% RSLogix 500 project WFETC_TOTS_R0.RSS, saved by version 12.00.00.00 %
PROJECT "WFETC"    % processor: SLC 500, 1747-L552 %

PROGRAM FILES
  LAD 2 "MAIN"  23 rungs
  LAD 3 "TE CONTROL"  1 rungs  % Set NT4 Input modules for Type J T/C's and °C Unit %
  LAD 4 "RIO BTRWS"  15 rungs  % Block Transfers for Remote IO %
  LAD 10 "ALARM CTRL"  9 rungs  % Alarm Controls %
  LAD 11 "ALARMS"  53 rungs  % Process Alarms %
  LAD 15 "IFIX PBS"  8 rungs  % iFIX PBs %
  LAD 16 "PV PBS"  11 rungs  % Panel View Screen Movement PB's %
  LAD 17 "VFD USERS"  17 rungs  % Determines which user is using each VFD %
  LAD 31 "MOVE TES"  20 rungs  % Move TE Info to Sequencial Locations, etc %
  LAD 32 "MOVE PTS"  7 rungs  % Move PT Info to Sequencial Locations, etc %
  LAD 33 "MOVE FTS"  6 rungs  % Move FT Info to Sequencial Locations, etc %
  LAD 34 "CALC WTS"  9 rungs  % Convert Remote I/O Data to Real Data for All Scale %
  LAD 35 "CALC WT FT"  10 rungs  % Calcualte Flow Rates based on Weight Changes %
  LAD 36 "CALC PTS"  15 rungs  % Calculate PT's Based on Max & Min Ranges %
  LAD 37 "CALC FTS"  8 rungs  % Calculate FT's Based on Max & Min Ranges %
  LAD 38 "CALC FYS"  35 rungs  % Calculate Flow Rates based on Scale Change & Time %
  LAD 39 "CALC ITS"  10 rungs  % Calculate SY Current Values %
  LAD 40 "CALC ATS"  7 rungs  % Calculate Densitys from FlowMeters %
  LAD 41 "CAL FTAVGS"  7 rungs  % Calculate FT Averages %
  LAD 42 "CALC LITS"  2 rungs  % Calculate LIT values %
  LAD 43 "CALLC TITS"  2 rungs  % Calculate TITs %
  LAD 48 "EF-1"  8 rungs  % Process Area Exhaust Fan Controls %
  LAD 49 "EF-2"  8 rungs  % Utility Room Exhaust Fan Controls %
  LAD 50 "EV-01"  8 rungs  % EV-1 Rotor Controls %
  LAD 51 "EV-02"  12 rungs  % EV-2 Rotor Drive VFD Controls %
  LAD 52 "EV-03"  12 rungs  % EV-3 Rotor Drive VFD Controls %
  LAD 53 "AG-04"  12 rungs  % AG-4 Agitator Drive VFD Controls %
  LAD 56 "VP-09"  8 rungs  % VP-9 Beach-Ross Vacuum Pump Controls %
  LAD 57 "VP-10"  8 rungs  % VP-10 Kinney Vacuum Pump Controls %
  LAD 60 "PU-11"  8 rungs  % PU-11 Tempered Water Loop No-1 Circ Pump Controls %
  LAD 61 "PU-12"  8 rungs  % PU-12 Tempered Water Loop No-2 Circ Pump Controls %
  LAD 62 "PU-15"  8 rungs  % PU-15 Tempered Oil Loop No-1 Circ Pump Controls %
  LAD 63 "EV-20"  12 rungs  % EV-20 Rotor Drive VFD Controls %
  LAD 64 "PU-21-1"  11 rungs  % PU-21-1 Feed Pump No-1 Controls %
  LAD 65 "PU-21-2"  11 rungs  % PU-21-2 Feed Pump No-2 Controls %
  LAD 66 "PU-21-3"  11 rungs  % PU-21-3 Feed Pump No-3 Controls %
  LAD 67 "PU-21-4"  11 rungs  % PU-21-4 Feed Pump No-4 Controls %
  LAD 69 "PU-22-1"  11 rungs  % PU-22-1 Level Pump No-1 Controls %
  LAD 71 "PU-23"  10 rungs  % PU-23 Hot Oil Circ Pump Controls %
  LAD 72 "EH-24"  7 rungs  % EH-24 Hot Oil Heater Controls %
  LAD 73 "VB-26"  9 rungs  % VB-26 Beach-Ross Vacuum Blower Controls %
  LAD 74 "PU-30"  9 rungs  % PU-30 Cooling Water Header Booster Pump Controls %
  LAD 75 "VB-35"  8 rungs  % VB-35 Tuthill Vacuum Blower Controls %
  LAD 77 "PU-37"  8 rungs  % PU-37, Temperaed Oil No-3 Controls %
  LAD 80 "PU-40"  8 rungs  % PU-40, Temperaed Oil No-2 Controls %
  LAD 81 "EV-42"  12 rungs  % EV-42 Rotor Drive VFD Controls %
  LAD 82 "PU-46"  11 rungs  % PU-46, Flash Evaporator Circ Pump %
  LAD 86 "ALL VFDS"  10 rungs  % Control All VFD's %
  LAD 90 "ALL PIDS"  17 rungs  % Execute All PID Statements using STI Interupt %
  LAD 101 "FIC-21-1"  12 rungs  % Feed Flow No-1 PID Controls %
  LAD 102 "FIC-21-2"  12 rungs  % Feed Flow No-2 PID Controls %
  LAD 103 "FIC-21-3"  12 rungs  % Feed Flow No-3 PID Controls %
  LAD 104 "FIC-21-4"  12 rungs  % Feed Flow No-4 PID Controls %
  LAD 111 "PIC-9-1"  14 rungs  % Vacuum Control No-1 PID %
  LAD 112 "PID-10-1"  14 rungs  % Vacuum Control No-2 PID %
  LAD 115 "PIC-28-1"  5 rungs  % Steam Pressure PID Controls %
  LAD 116 "PIC-30-1"  6 rungs  % Cooling Water Pressure PID Controls %
  LAD 117 "PIC-46-1"  6 rungs  % Flash Evap Pressure Controller %
  LAD 121 "TIC-11-1"  6 rungs  % Tempered Water Loop No-1 Temperature PID Controls %
  LAD 122 "TIC-12-1"  7 rungs  % Tempered Water Loop No-2 Temperature PID Controls %
  LAD 123 "TIC-15-1"  6 rungs  % Tempered Oil Loop No-1 Temperature PID Controls %
  LAD 124 "TIC-24-1"  6 rungs  % Hot Oil Temperature PID Controls %
  LAD 125 "TIC-37-1"  6 rungs  % Tempered Oil Loop No-3 Temperature PID Controls %
  LAD 126 "TIC-40-1"  6 rungs  % Tempered Oil Loop No-2 Temperature PID Controls %
  LAD 131 "LIC-22-1"  7 rungs  % Level Control No-1 PID Controls %
  LAD 132 "TOTALIZER"  8 rungs

DATA FILES
  O0 OUTPUT  99 elements
  I1 INPUT  111 elements
  S2 STATUS  83 elements
  B3 BINARY  81 elements
  T4 TIMER  36 elements
  C5 COUNTER  15 elements
  R6 CONTROL  1 elements
  N7 INTEGER  23 elements
  F8 FLOAT  256 elements
  N11 AI INTEGER  250 elements  % Integer Data for All Inputs (TE's, PT's and FT's) %
  N12 RIO DATA  200 elements  % Remote I/O Data %
  N13 TE SETUP  200 elements  % TE Setup Data %
  F14 SETPOINTS  100 elements  % Setpoints for various Alarms, trips, etc %
  N15 PID 1 OF 3  240 elements  % PID Statement Controls File No-1 %
  N16 PID 2 OF 3  175 elements  % PID Statement Controls File No-2 %
  N17 PID 3 OF 3  180 elements  % PID Statement Controls File No-3 %
  N18 PID OUTPUT  60 elements  % Outputs from All PID Statements %
  N20 PANELVIEW  100 elements  % Info From/to PanelView HMIs %
  F21 AI REAL  256 elements
  F22 AI BY TAG  250 elements
  N23 AI PTRS  256 elements
  N24 FIXED INTS  250 elements  % Fixed Integer Values %
  N25 VAR INTS  200 elements  % Variable Integer Values %
  F26 FIXEDREAL1  250 elements  % Fixed Real (Floating Point) Data 1 of 2 %
  F27 VAR REAL  210 elements  % Variable Real (Floatinf Point) Data %
  F28 FLOW AVGS  51 elements  % Flow Data used to Calculate 5 Minute Aveerages %
  F29 PID PCNTS1  250 elements  % PID Statement 0, 25, 50, 75 & 100% Values %
  F30 FIXEDREAL2  250 elements  % Fixed Real (Floating Point) Data 2 of 2 %
  F31 PID PCNTS2  220 elements
  N50 CNTL BITS  50 elements  % Control Bits for all Motors, Contacters, Etc %
  T51 ALARM TMRS  100 elements  % Alarm Timers %
  F52 ALARM SPS  50 elements  % Alarm Setpoints %
  F60 VFD TABLE  50 elements  % Provide sequencial table for VFD outputs %
  N61 VFD BITS  10 elements  % Provide seq table for VFD Contrl & Status Bits %
  F62 VFD AMPS  10 elements  % VFD Amps %
  F63 VFD HP  20 elements  % Motor and VFD Hps %
  N100 CH0 Diag  32 elements
  N101 CH1 Diag  256 elements
  F201 FT1 AVGS  51 elements  % Average FT-1 Values %
  F202 FT2 AVGS  51 elements  % Average FT-2 Values %
  F203 FT3 AVGS  51 elements  % Average FT-3 Values %
  F204 FT4 AVGS  51 elements  % Average FT-4 Values %
  F205 FT5 AVGS  51 elements  % Average FT-5 Values %
  F206 FT6 AVGS  51 elements  % Average FT-6 Values %

LADDER 2 "MAIN"
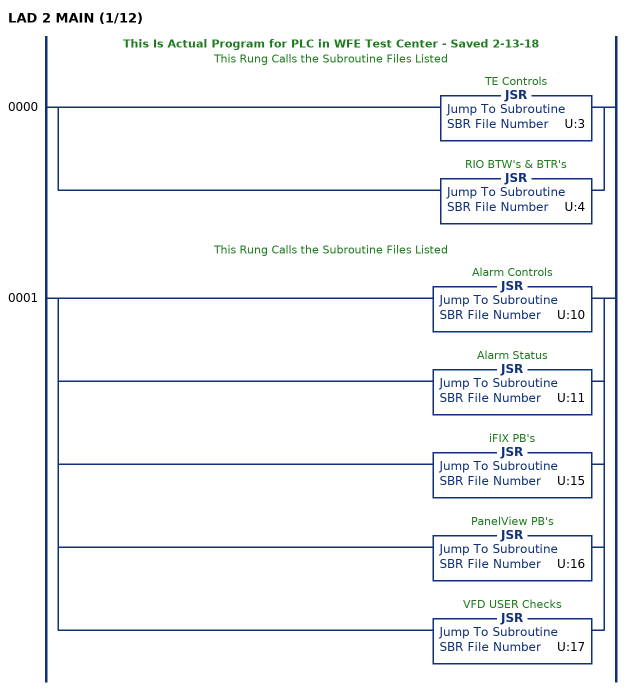
% Rung: 0 %
% TITLE: This Is Actual Program for PLC in WFE Test Center - Saved 2-13-18 %
% This Rung Calls the Subroutine Files Listed %
SOR BST JSR U:3 NXB JSR U:4 BND EOR
%   U:3  "TE Controls" %
%   U:4  "RIO BTW's & BTR's" %
% Rung: 1 %
% This Rung Calls the Subroutine Files Listed %
SOR BST JSR U:10 NXB JSR U:11 NXB JSR U:15 NXB JSR U:16 NXB JSR U:17 BND EOR
%   U:10  "Alarm Controls" %
%   U:11  "Alarm Status" %
%   U:15  "iFIX PB's" %
%   U:16  "PanelView PB's" %
%   U:17  "VFD USER Checks" %

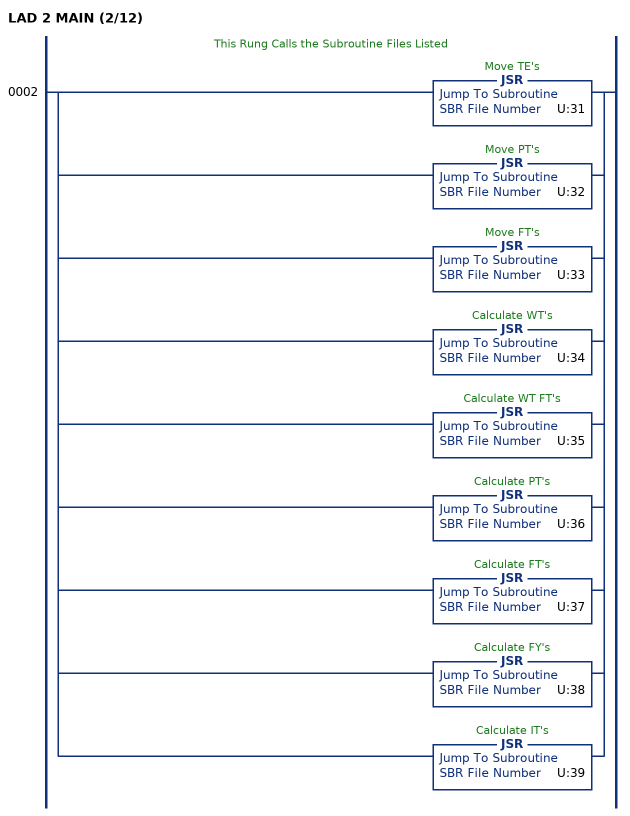
% Rung: 2 %
% This Rung Calls the Subroutine Files Listed %
SOR BST JSR U:31 NXB JSR U:32 NXB JSR U:33 NXB JSR U:34 NXB JSR U:35 NXB JSR U:36 NXB JSR U:37 NXB JSR U:38 NXB JSR U:39 BND EOR
%   U:31  "Move TE's" %
%   U:32  "Move PT's" %
%   U:33  "Move FT's" %
%   U:34  "Calculate WT's" %
%   U:35  "Calculate WT FT's" %
%   U:36  "Calculate PT's" %
%   U:37  "Calculate FT's" %
%   U:38  "Calculate FY's" %
%   U:39  "Calculate IT's" %

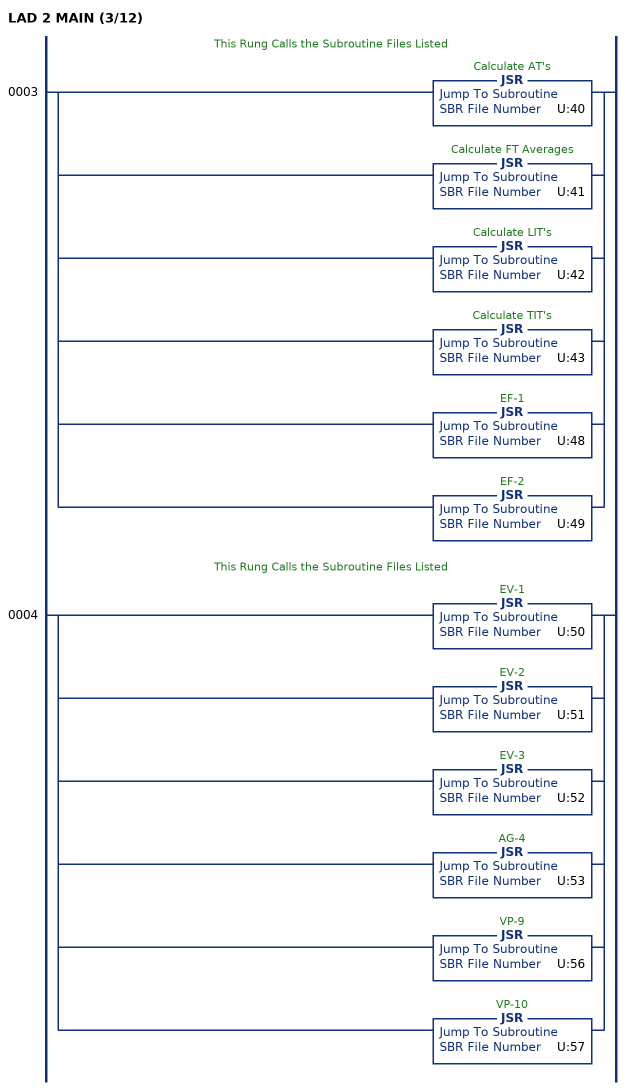
% Rung: 3 %
% This Rung Calls the Subroutine Files Listed %
SOR BST JSR U:40 NXB JSR U:41 NXB JSR U:42 NXB JSR U:43 NXB JSR U:48 NXB JSR U:49 BND EOR
%   U:40  "Calculate AT's" %
%   U:41  "Calculate FT Averages" %
%   U:42  "Calculate LIT's" %
%   U:43  "Calculate TIT's" %
%   U:48  "EF-1" %
%   U:49  "EF-2" %
% Rung: 4 %
% This Rung Calls the Subroutine Files Listed %
SOR BST JSR U:50 NXB JSR U:51 NXB JSR U:52 NXB JSR U:53 NXB JSR U:56 NXB JSR U:57 BND EOR
%   U:50  "EV-1" %
%   U:51  "EV-2" %
%   U:52  "EV-3" %
%   U:53  "AG-4" %
%   U:56  "VP-9" %
%   U:57  "VP-10" %

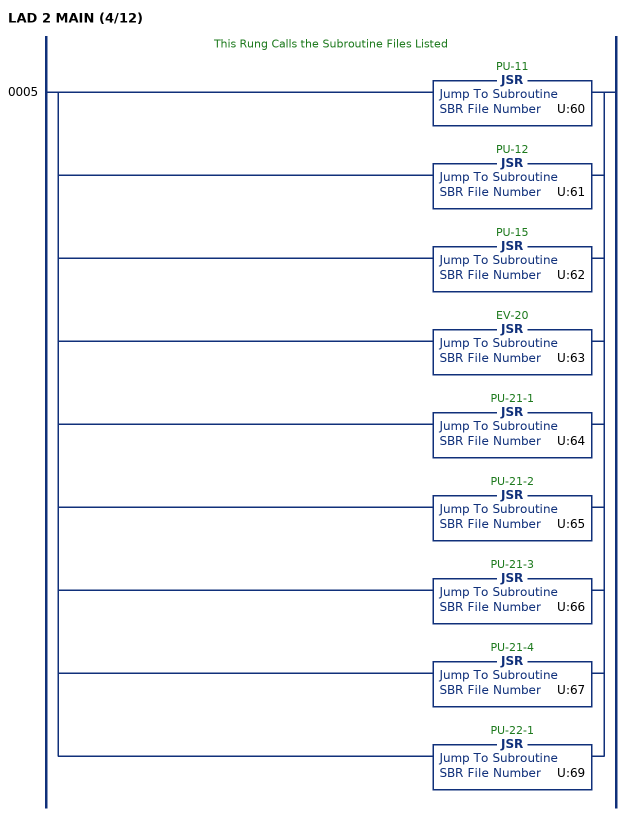
% Rung: 5 %
% This Rung Calls the Subroutine Files Listed %
SOR BST JSR U:60 NXB JSR U:61 NXB JSR U:62 NXB JSR U:63 NXB JSR U:64 NXB JSR U:65 NXB JSR U:66 NXB JSR U:67 NXB JSR U:69 BND EOR
%   U:60  "PU-11" %
%   U:61  "PU-12" %
%   U:62  "PU-15" %
%   U:63  "EV-20" %
%   U:64  "PU-21-1" %
%   U:65  "PU-21-2" %
%   U:66  "PU-21-3" %
%   U:67  "PU-21-4" %
%   U:69  "PU-22-1" %

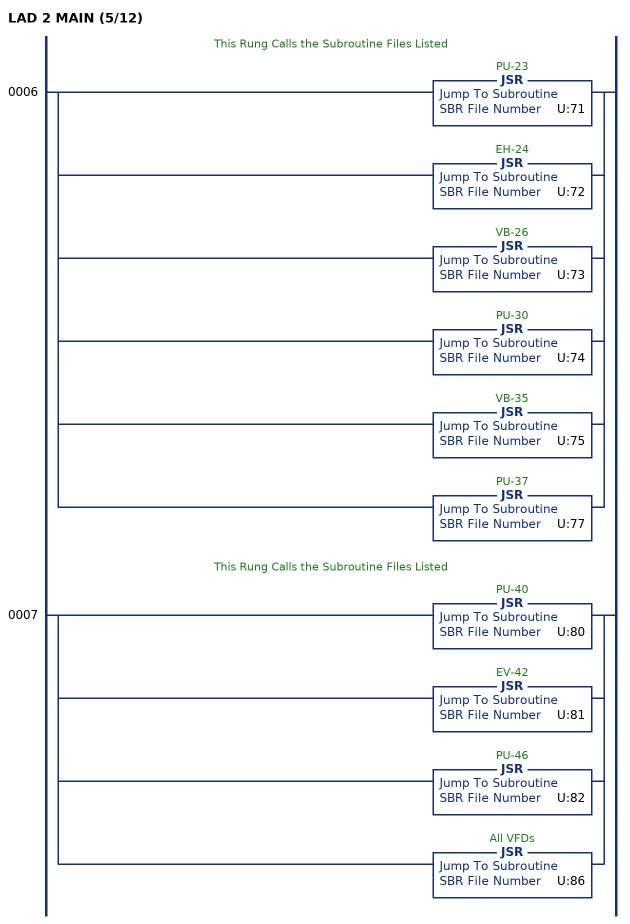
% Rung: 6 %
% This Rung Calls the Subroutine Files Listed %
SOR BST JSR U:71 NXB JSR U:72 NXB JSR U:73 NXB JSR U:74 NXB JSR U:75 NXB JSR U:77 BND EOR
%   U:71  "PU-23" %
%   U:72  "EH-24" %
%   U:73  "VB-26" %
%   U:74  "PU-30" %
%   U:75  "VB-35" %
%   U:77  "PU-37" %
% Rung: 7 %
% This Rung Calls the Subroutine Files Listed %
SOR BST JSR U:80 NXB JSR U:81 NXB JSR U:82 NXB JSR U:86 BND EOR
%   U:80  "PU-40" %
%   U:81  "EV-42" %
%   U:82  "PU-46" %
%   U:86  "All VFDs" %

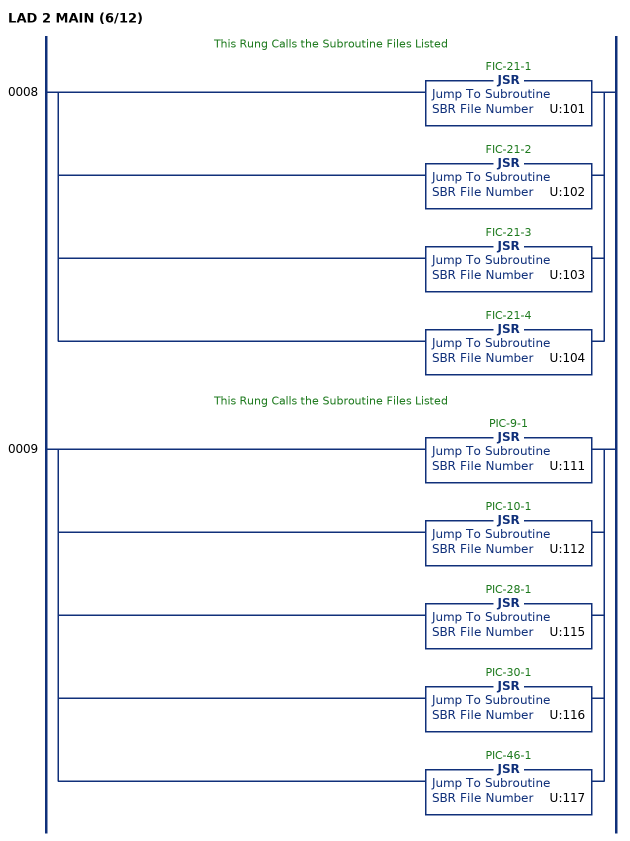
% Rung: 8 %
% This Rung Calls the Subroutine Files Listed %
SOR BST JSR U:101 NXB JSR U:102 NXB JSR U:103 NXB JSR U:104 BND EOR
%   U:101  "FIC-21-1" %
%   U:102  "FIC-21-2" %
%   U:103  "FIC-21-3" %
%   U:104  "FIC-21-4" %
% Rung: 9 %
% This Rung Calls the Subroutine Files Listed %
SOR BST JSR U:111 NXB JSR U:112 NXB JSR U:115 NXB JSR U:116 NXB JSR U:117 BND EOR
%   U:111  "PIC-9-1" %
%   U:112  "PIC-10-1" %
%   U:115  "PIC-28-1" %
%   U:116  "PIC-30-1" %
%   U:117  "PIC-46-1" %

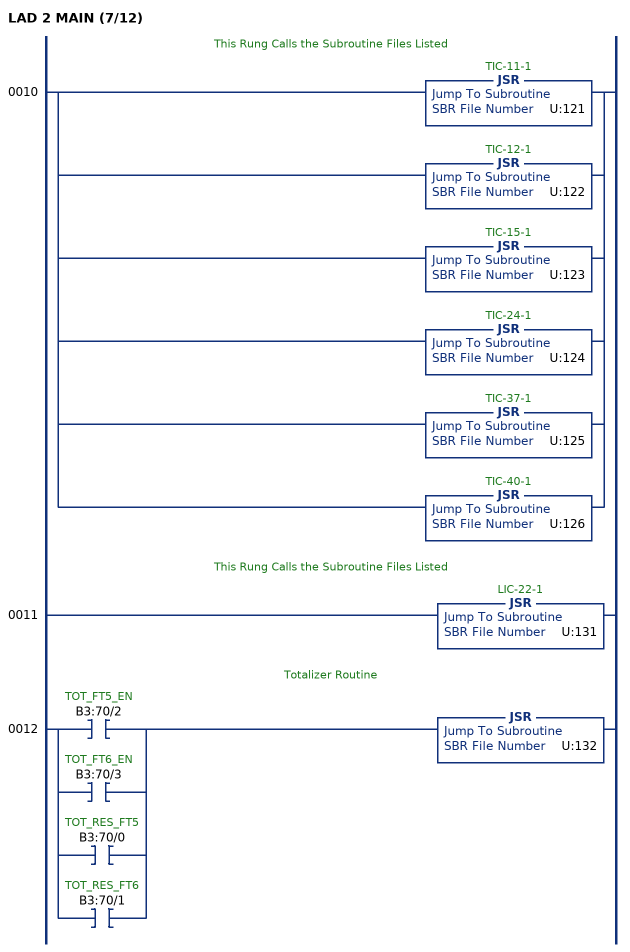
% Rung: 10 %
% This Rung Calls the Subroutine Files Listed %
SOR BST JSR U:121 NXB JSR U:122 NXB JSR U:123 NXB JSR U:124 NXB JSR U:125 NXB JSR U:126 BND EOR
%   U:121  "TIC-11-1" %
%   U:122  "TIC-12-1" %
%   U:123  "TIC-15-1" %
%   U:124  "TIC-24-1" %
%   U:125  "TIC-37-1" %
%   U:126  "TIC-40-1" %
% Rung: 11 %
% This Rung Calls the Subroutine Files Listed %
SOR JSR U:131 EOR
%   U:131  "LIC-22-1" %
% Rung: 12 %
% Totalizer Routine %
SOR BST XIC B3:70/2 NXB BST XIC B3:70/3 NXB BST XIC B3:70/0 NXB XIC B3:70/1 BND BND BND JSR U:132 EOR
%   B3:70/2  TOT_FT5_EN %
%   B3:70/3  TOT_FT6_EN %
%   B3:70/0  TOT_RES_FT5 %
%   B3:70/1  TOT_RES_FT6 %

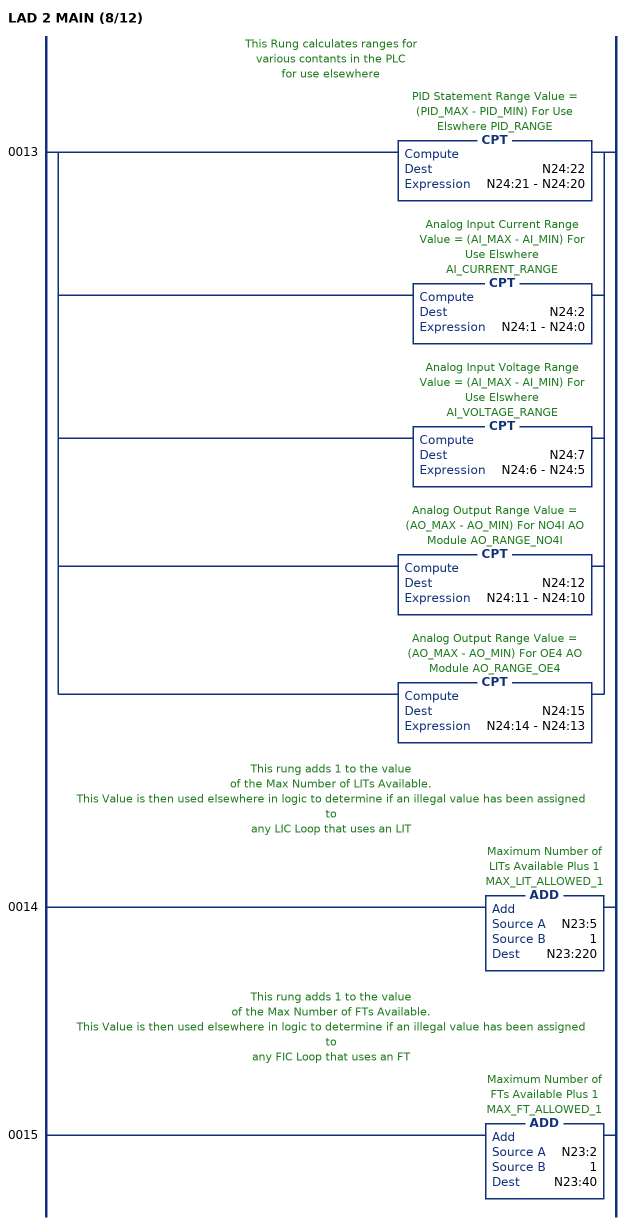
% Rung: 13 %
% This Rung calculates ranges for
% various contants in the PLC
% for use elsewhere %
SOR BST CPT N24:22 " N24:21 - N24:20 " NXB CPT N24:2 " N24:1 - N24:0 " NXB CPT N24:7 " N24:6 - N24:5 " NXB CPT N24:12 " N24:11 - N24:10 " NXB CPT N24:15 " N24:14 - N24:13 " BND EOR
%   N24:22  PID_RANGE  "PID Statement Range Value = (PID_MAX - PID_MIN) For Use Elswhere" %
%   N24:21  PID_MAX  "PID Statement Maximum Value" %
%   N24:20  PID_MIN  "PID Statement Minimum Value" %
%   N24:2  AI_CURRENT_RANGE  "Analog Input Current Range Value = (AI_MAX - AI_MIN) For Use Elswhere" %
%   N24:1  AI_CURRENT_MAX  "Analog Input Maximum Value = 20 mA DC (From AI Module)" %
%   N24:0  AI_CURRENT_MIN  "Analog Input Minimum Value = 4 mA DC (From AI Module)" %
%   N24:7  AI_VOLTAGE_RANGE  "Analog Input Voltage Range Value = (AI_MAX - AI_MIN) For Use Elswhere" %
%   N24:6  AI_VOLTAGE_MAX  "Analog Input Maximum Value = 10 VDC (From AI Module)" %
%   N24:5  AI_VOLTAGE_MIN  "Analog Input Minimum Value = 0 VDC (From AI Module)" %
%   N24:12  AO_RANGE_NO4I  "Analog Output Range Value = (AO_MAX - AO_MIN) For NO4I AO Module" %
%   N24:11  AO_MAX_NO4I  "Analog Output Maximum Value Generates 20 mA DC (To NO4I AO Module)" %
%   N24:10  AO_MIN_NO4I  "Analog Output Minimum Value Generates 4 mA DC (To NO4I AO Module)" %
%   N24:15  AO_RANGE_OE4  "Analog Output Range Value = (AO_MAX - AO_MIN) For OE4 AO Module" %
%   N24:14  AO_MAX_OE4  "Analog Output Maximum Value Generates 20 mA DC (To OE4 AO Module)" %
%   N24:13  AO_MIN_OE4  "Analog Output Minimum Value Generates 4 mA DC (To OE4 AO Module)" %
% Rung: 14 %
% This rung adds 1 to the value
% of the Max Number of LITs Available.
% This Value is then used elsewhere in logic to determine if an illegal value has been assigned to
% any LIC Loop that uses an LIT %
SOR ADD N23:5 1 N23:220 EOR
%   N23:5  LIT_PTR_MAX  "Maximum Value for LIT Pointer" %
%   N23:220  MAX_LIT_ALLOWED_1  "Maximum Number of LITs Available Plus 1" %
% Rung: 15 %
% This rung adds 1 to the value
% of the Max Number of FTs Available.
% This Value is then used elsewhere in logic to determine if an illegal value has been assigned to
% any FIC Loop that uses an FT %
SOR ADD N23:2 1 N23:40 EOR
%   N23:2  FT_PTR_MAX  "Maximum Value for FT Pointer" %
%   N23:40  MAX_FT_ALLOWED_1  "Maximum Number of FTs Available Plus 1" %

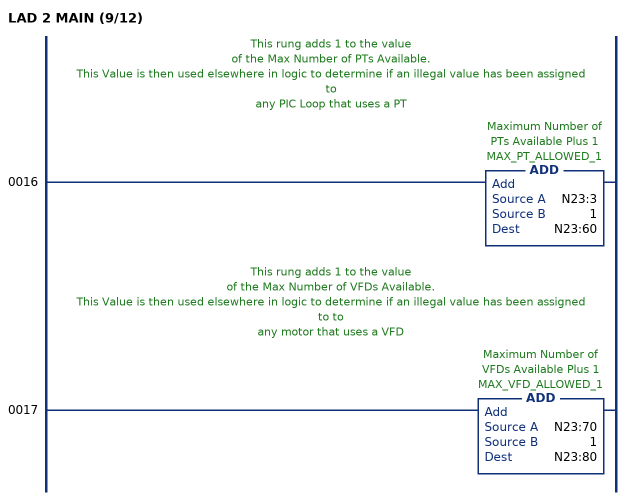
% Rung: 16 %
% This rung adds 1 to the value
% of the Max Number of PTs Available.
% This Value is then used elsewhere in logic to determine if an illegal value has been assigned to
% any PIC Loop that uses a PT %
SOR ADD N23:3 1 N23:60 EOR
%   N23:3  PT_PTR_MAX  "Maximum Value for PT Pointer" %
%   N23:60  MAX_PT_ALLOWED_1  "Maximum Number of PTs Available Plus 1" %
% Rung: 17 %
% This rung adds 1 to the value
% of the Max Number of VFDs Available.
% This Value is then used elsewhere in logic to determine if an illegal value has been assigned to to
% any motor that uses a VFD %
SOR ADD N23:70 1 N23:80 EOR
%   N23:70  MAX_VFD_ALLOWED  "Maximum Number of VFDs Available" %
%   N23:80  MAX_VFD_ALLOWED_1  "Maximum Number of VFDs Available Plus 1" %

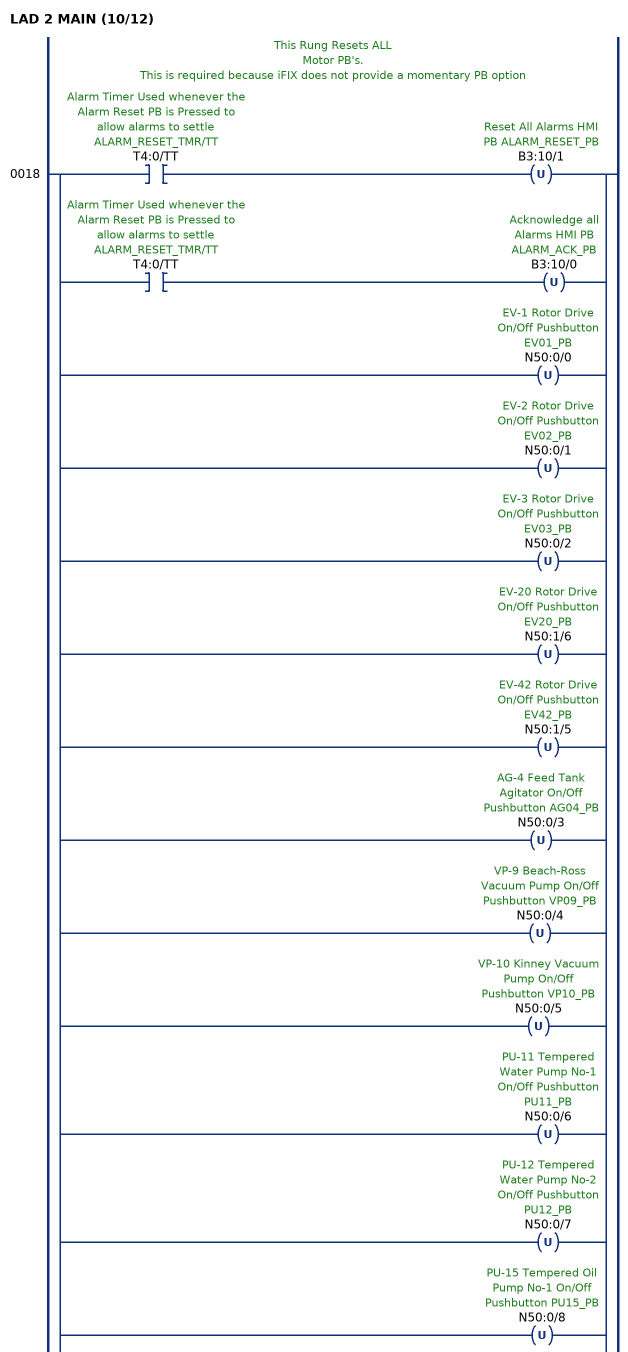

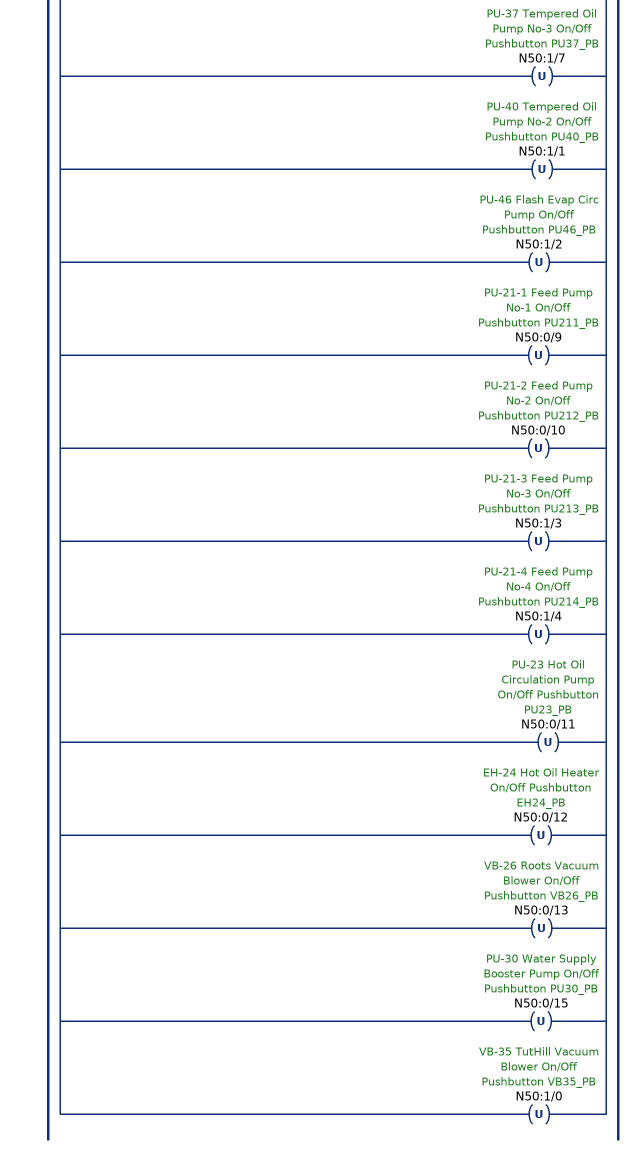
% Rung: 18 %
% This Rung Resets ALL
% Motor PB's.
% This is required because iFIX does not provide a momentary PB option %
SOR BST XIC T4:0/TT OTU B3:10/1 NXB XIC T4:0/TT OTU B3:10/0 NXB OTU N50:0/0 NXB OTU N50:0/1 NXB OTU N50:0/2 NXB OTU N50:1/6 NXB OTU N50:1/5 NXB OTU N50:0/3 NXB OTU N50:0/4 NXB OTU N50:0/5 NXB OTU N50:0/6 NXB OTU N50:0/7 NXB OTU N50:0/8 NXB OTU N50:1/7 NXB OTU N50:1/1 NXB OTU N50:1/2 NXB OTU N50:0/9 NXB OTU N50:0/10 NXB OTU N50:1/3 NXB OTU N50:1/4 NXB OTU N50:0/11 NXB OTU N50:0/12 NXB OTU N50:0/13 NXB OTU N50:0/15 NXB OTU N50:1/0 BND EOR
%   T4:0  ALARM_RESET_TMR  "Alarm Timer Used whenever the Alarm Reset PB is Pressed to allow alarms to settle" %
%   B3:10/1  ALARM_RESET_PB  "Reset All Alarms HMI PB" %
%   B3:10/0  ALARM_ACK_PB  "Acknowledge all Alarms HMI PB" %
%   N50:0/0  EV01_PB  "EV-1 Rotor Drive On/Off Pushbutton" %
%   N50:0/1  EV02_PB  "EV-2 Rotor Drive On/Off Pushbutton" %
%   N50:0/2  EV03_PB  "EV-3 Rotor Drive On/Off Pushbutton" %
%   N50:1/6  EV20_PB  "EV-20 Rotor Drive On/Off Pushbutton" %
%   N50:1/5  EV42_PB  "EV-42 Rotor Drive On/Off Pushbutton" %
%   N50:0/3  AG04_PB  "AG-4 Feed Tank Agitator On/Off Pushbutton" %
%   N50:0/4  VP09_PB  "VP-9 Beach-Ross Vacuum Pump On/Off Pushbutton" %
%   N50:0/5  VP10_PB  "VP-10 Kinney Vacuum Pump On/Off Pushbutton" %
%   N50:0/6  PU11_PB  "PU-11 Tempered Water Pump No-1 On/Off Pushbutton" %
%   N50:0/7  PU12_PB  "PU-12 Tempered Water Pump No-2 On/Off Pushbutton" %
%   N50:0/8  PU15_PB  "PU-15 Tempered Oil Pump No-1 On/Off Pushbutton" %
%   N50:1/7  PU37_PB  "PU-37 Tempered Oil Pump No-3 On/Off Pushbutton" %
%   N50:1/1  PU40_PB  "PU-40 Tempered Oil Pump No-2 On/Off Pushbutton" %
%   N50:1/2  PU46_PB  "PU-46 Flash Evap Circ Pump On/Off Pushbutton" %
%   N50:0/9  PU211_PB  "PU-21-1 Feed Pump No-1 On/Off Pushbutton" %
%   N50:0/10  PU212_PB  "PU-21-2 Feed Pump No-2 On/Off Pushbutton" %
%   N50:1/3  PU213_PB  "PU-21-3 Feed Pump No-3 On/Off Pushbutton" %
%   N50:1/4  PU214_PB  "PU-21-4 Feed Pump No-4 On/Off Pushbutton" %
%   N50:0/11  PU23_PB  "PU-23 Hot Oil Circulation Pump On/Off Pushbutton" %
%   N50:0/12  EH24_PB  "EH-24 Hot Oil Heater On/Off Pushbutton" %
%   N50:0/13  VB26_PB  "VB-26 Roots Vacuum Blower On/Off Pushbutton" %
%   N50:0/15  PU30_PB  "PU-30 Water Supply Booster Pump On/Off Pushbutton" %
%   N50:1/0  VB35_PB  "VB-35 TutHill Vacuum Blower On/Off Pushbutton" %

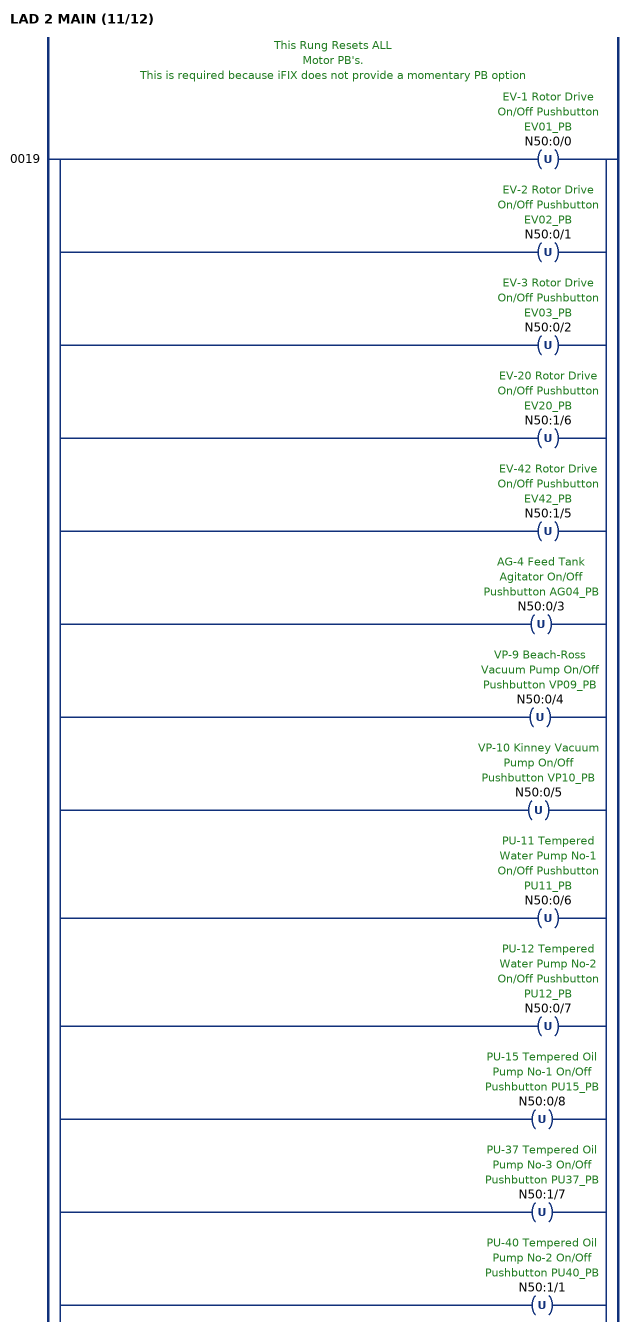

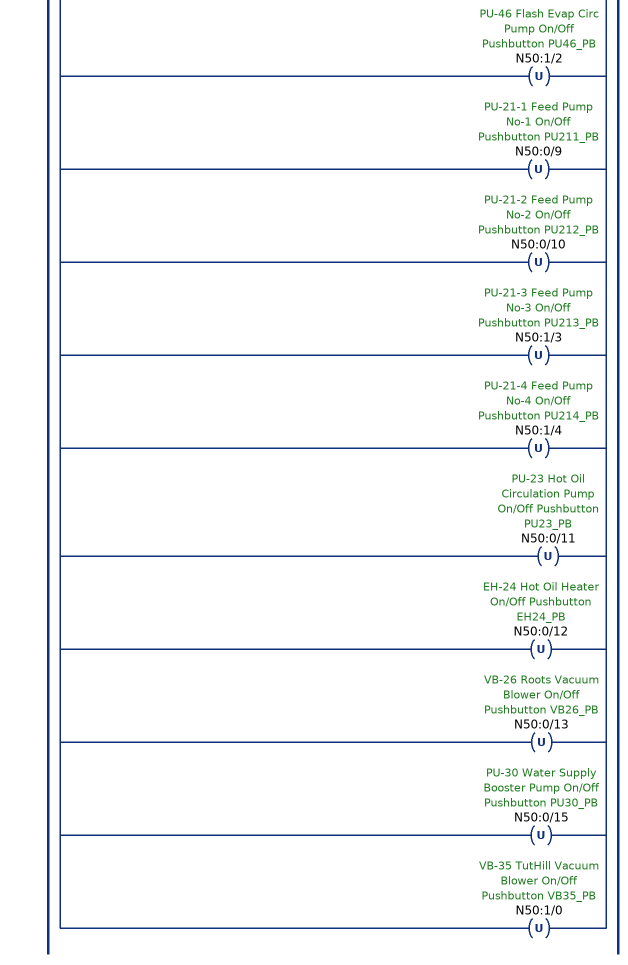
% Rung: 19 %
% This Rung Resets ALL
% Motor PB's.
% This is required because iFIX does not provide a momentary PB option %
SOR BST OTU N50:0/0 NXB OTU N50:0/1 NXB OTU N50:0/2 NXB OTU N50:1/6 NXB OTU N50:1/5 NXB OTU N50:0/3 NXB OTU N50:0/4 NXB OTU N50:0/5 NXB OTU N50:0/6 NXB OTU N50:0/7 NXB OTU N50:0/8 NXB OTU N50:1/7 NXB OTU N50:1/1 NXB OTU N50:1/2 NXB OTU N50:0/9 NXB OTU N50:0/10 NXB OTU N50:1/3 NXB OTU N50:1/4 NXB OTU N50:0/11 NXB OTU N50:0/12 NXB OTU N50:0/13 NXB OTU N50:0/15 NXB OTU N50:1/0 BND EOR
%   N50:0/0  EV01_PB  "EV-1 Rotor Drive On/Off Pushbutton" %
%   N50:0/1  EV02_PB  "EV-2 Rotor Drive On/Off Pushbutton" %
%   N50:0/2  EV03_PB  "EV-3 Rotor Drive On/Off Pushbutton" %
%   N50:1/6  EV20_PB  "EV-20 Rotor Drive On/Off Pushbutton" %
%   N50:1/5  EV42_PB  "EV-42 Rotor Drive On/Off Pushbutton" %
%   N50:0/3  AG04_PB  "AG-4 Feed Tank Agitator On/Off Pushbutton" %
%   N50:0/4  VP09_PB  "VP-9 Beach-Ross Vacuum Pump On/Off Pushbutton" %
%   N50:0/5  VP10_PB  "VP-10 Kinney Vacuum Pump On/Off Pushbutton" %
%   N50:0/6  PU11_PB  "PU-11 Tempered Water Pump No-1 On/Off Pushbutton" %
%   N50:0/7  PU12_PB  "PU-12 Tempered Water Pump No-2 On/Off Pushbutton" %
%   N50:0/8  PU15_PB  "PU-15 Tempered Oil Pump No-1 On/Off Pushbutton" %
%   N50:1/7  PU37_PB  "PU-37 Tempered Oil Pump No-3 On/Off Pushbutton" %
%   N50:1/1  PU40_PB  "PU-40 Tempered Oil Pump No-2 On/Off Pushbutton" %
%   N50:1/2  PU46_PB  "PU-46 Flash Evap Circ Pump On/Off Pushbutton" %
%   N50:0/9  PU211_PB  "PU-21-1 Feed Pump No-1 On/Off Pushbutton" %
%   N50:0/10  PU212_PB  "PU-21-2 Feed Pump No-2 On/Off Pushbutton" %
%   N50:1/3  PU213_PB  "PU-21-3 Feed Pump No-3 On/Off Pushbutton" %
%   N50:1/4  PU214_PB  "PU-21-4 Feed Pump No-4 On/Off Pushbutton" %
%   N50:0/11  PU23_PB  "PU-23 Hot Oil Circulation Pump On/Off Pushbutton" %
%   N50:0/12  EH24_PB  "EH-24 Hot Oil Heater On/Off Pushbutton" %
%   N50:0/13  VB26_PB  "VB-26 Roots Vacuum Blower On/Off Pushbutton" %
%   N50:0/15  PU30_PB  "PU-30 Water Supply Booster Pump On/Off Pushbutton" %
%   N50:1/0  VB35_PB  "VB-35 TutHill Vacuum Blower On/Off Pushbutton" %

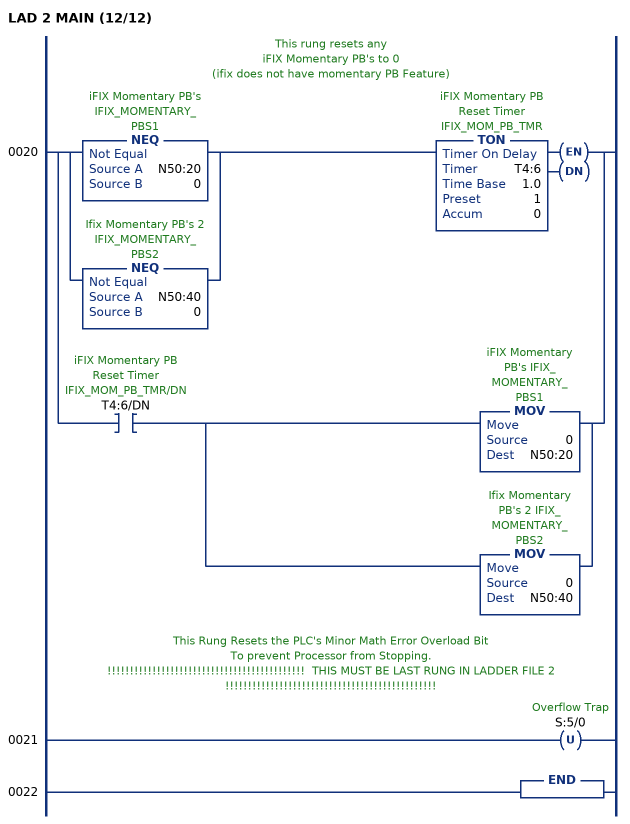
% Rung: 20 %
% This rung resets any
% iFIX Momentary PB's to 0
% (ifix does not have momentary PB Feature) %
SOR BST BST NEQ N50:20 0 NXB NEQ N50:40 0 BND TON T4:6 1.0 1 0 NXB XIC T4:6/DN BST MOV 0 N50:20 NXB MOV 0 N50:40 BND BND EOR
%   N50:20  IFIX_MOMENTARY_PBS1  "iFIX Momentary PB's" %
%   N50:40  IFIX_MOMENTARY_PBS2  "Ifix Momentary PB's 2" %
%   T4:6  IFIX_MOM_PB_TMR  "iFIX Momentary PB Reset Timer" %
% Rung: 21 %
% This Rung Resets the PLC's Minor Math Error Overload Bit
% To prevent Processor from Stopping.
% !!!!!!!!!!!!!!!!!!!!!!!!!!!!!!!!!!!!!!!!!!!!  THIS MUST BE LAST RUNG IN LADDER FILE 2 !!!!!!!!!!!!!!!!!!!!!!!!!!!!!!!!!!!!!!!!!!!!!!! %
SOR OTU S:5/0 EOR
%   S:5/0  "Overflow Trap" %
% Rung: 22 %
SOR END EOR

LADDER 4 "RIO BTRWS"    % Block Transfers for Remote IO %
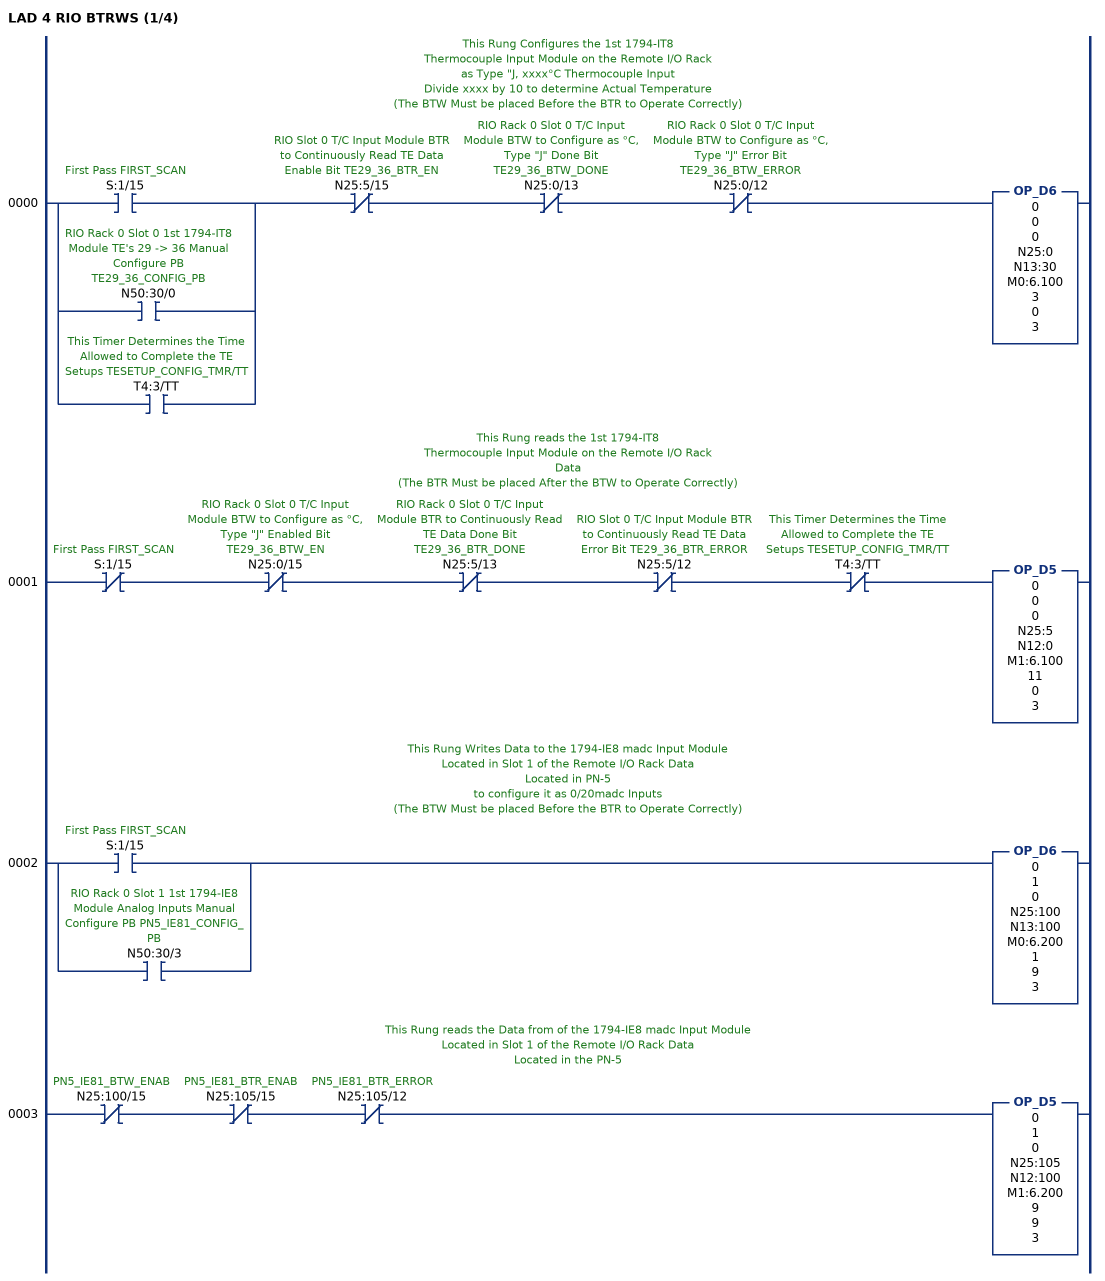
% Rung: 0 %
% This Rung Configures the 1st 1794-IT8
% Thermocouple Input Module on the Remote I/O Rack
% as Type "J, xxxx°C Thermocouple Input
% Divide xxxx by 10 to determine Actual Temperature
% 
% (The BTW Must be placed Before the BTR to Operate Correctly) %
SOR BST XIC S:1/15 NXB XIC N50:30/0 NXB XIC T4:3/TT BND XIO N25:5/15 XIO N25:0/13 XIO N25:0/12 OP_D6 0 0 0 N25:0 N13:30 M0:6.100 3 0 3 EOR
%   S:1/15  FIRST_SCAN  "First Pass" %
%   N50:30/0  TE29_36_CONFIG_PB  "RIO Rack 0 Slot 0 1st 1794-IT8 Module TE's 29 -> 36 Manual Configure PB" %
%   T4:3  TESETUP_CONFIG_TMR  "This Timer Determines the Time Allowed to Complete the TE Setups" %
%   N25:5/15  TE29_36_BTR_EN  "RIO Slot 0 T/C Input Module BTR to Continuously Read TE Data Enable Bit" %
%   N25:0/13  TE29_36_BTW_DONE  "RIO Rack 0 Slot 0 T/C Input Module BTW to Configure as °C, Type "J" Done Bit" %
%   N25:0/12  TE29_36_BTW_ERROR  "RIO Rack 0 Slot 0 T/C Input Module BTW to Configure as °C, Type "J" Error Bit" %
%   N25:0  TE29_36_BTW_WORD_0  "RIO Rack 0 Slot 0 T/C Input Module BTW to Configure as °C, Type "J"" %
%   N13:30  TE29_36_SETUP_WORD_0  "RIO 1794-IT8 Setup Word 0 Set Units to °C" %
% Rung: 1 %
% This Rung reads the 1st 1794-IT8
% Thermocouple Input Module on the Remote I/O Rack
% Data
% 
% (The BTR Must be placed After the BTW to Operate Correctly) %
SOR XIO S:1/15 XIO N25:0/15 XIO N25:5/13 XIO N25:5/12 XIO T4:3/TT OP_D5 0 0 0 N25:5 N12:0 M1:6.100 11 0 3 EOR
%   S:1/15  FIRST_SCAN  "First Pass" %
%   N25:0/15  TE29_36_BTW_EN  "RIO Rack 0 Slot 0 T/C Input Module BTW to Configure as °C, Type "J" Enabled Bit" %
%   N25:5/13  TE29_36_BTR_DONE  "RIO Rack 0 Slot 0 T/C Input Module BTR to Continuously Read TE Data Done Bit" %
%   N25:5/12  TE29_36_BTR_ERROR  "RIO Slot 0 T/C Input Module BTR to Continuously Read TE Data Error Bit" %
%   T4:3  TESETUP_CONFIG_TMR  "This Timer Determines the Time Allowed to Complete the TE Setups" %
%   N25:5  TE29_36_BTR_WORD_0  "RIO Rack 0 Slot 0 T/C Input Module BTR to Continuously Read TE Data" %
%   N12:0  TE29_36_BTR_DATA0  "TE-29 thru TE-36 BTR Data 1" %
% Rung: 2 %
% This Rung Writes Data to the 1794-IE8 madc Input Module
% Located in Slot 1 of the Remote I/O Rack Data
% Located in PN-5
% to configure it as 0/20madc Inputs
% 
% (The BTW Must be placed Before the BTR to Operate Correctly) %
SOR BST XIC S:1/15 NXB XIC N50:30/3 BND OP_D6 0 1 0 N25:100 N13:100 M0:6.200 1 9 3 EOR
%   S:1/15  FIRST_SCAN  "First Pass" %
%   N50:30/3  PN5_IE81_CONFIG_PB  "RIO Rack 0 Slot 1 1st 1794-IE8 Module Analog Inputs Manual Configure PB" %
%   N25:100  PN5_IE81_BTW_WORD_0  "RIO Rack 0 Slot 1 Analog Input Module BTW to Update Data to Outputs Word 0" %
%   N13:100  PN5_IE81_BTW_DATA  "PN5 RIO Slot 1 Input Configuration Data ma = 0/20madc VDV = 0/10VDV" %
% Rung: 3 %
% This Rung reads the Data from of the 1794-IE8 madc Input Module
% Located in Slot 1 of the Remote I/O Rack Data
% Located in the PN-5 %
SOR XIO N25:100/15 XIO N25:105/15 XIO N25:105/12 OP_D5 0 1 0 N25:105 N12:100 M1:6.200 9 9 3 EOR
%   N25:100/15  PN5_IE81_BTW_ENAB %
%   N25:105/15  PN5_IE81_BTR_ENAB %
%   N25:105/12  PN5_IE81_BTR_ERROR %
%   N25:105  PN5_IE81_BTR_WORD_0  "RIO Rack 0 Slot 1 Analog Input Module BTR to Read Data Word 0" %
%   N12:100  AI101_BIN_DATA %

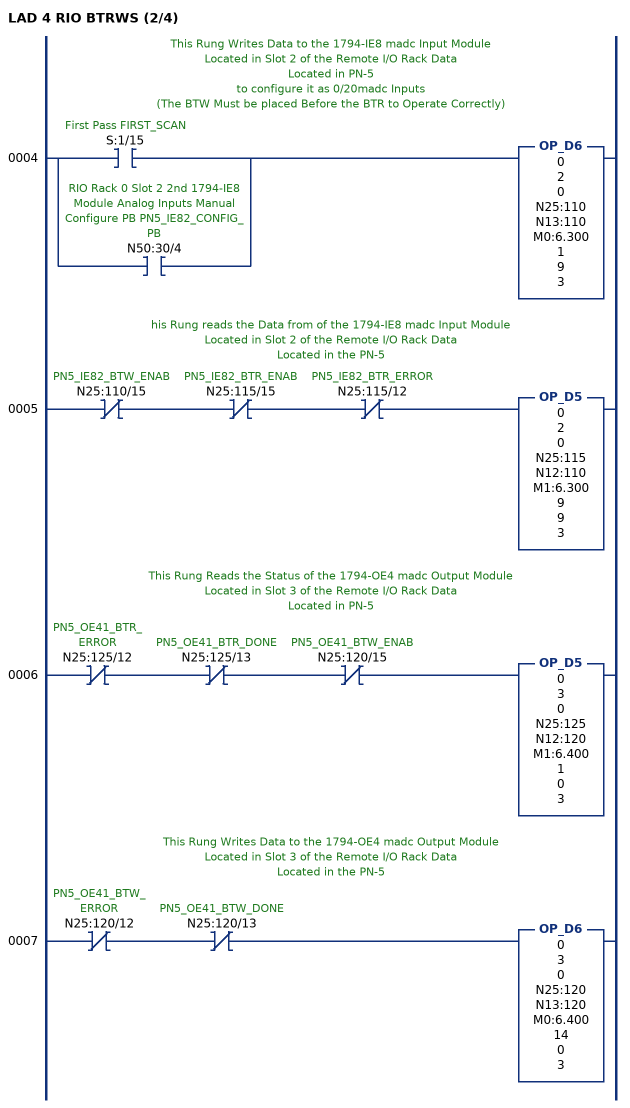
% Rung: 4 %
% This Rung Writes Data to the 1794-IE8 madc Input Module
% Located in Slot 2 of the Remote I/O Rack Data
% Located in PN-5
% to configure it as 0/20madc Inputs
% 
% (The BTW Must be placed Before the BTR to Operate Correctly) %
SOR BST XIC S:1/15 NXB XIC N50:30/4 BND OP_D6 0 2 0 N25:110 N13:110 M0:6.300 1 9 3 EOR
%   S:1/15  FIRST_SCAN  "First Pass" %
%   N50:30/4  PN5_IE82_CONFIG_PB  "RIO Rack 0 Slot 2 2nd 1794-IE8 Module Analog Inputs Manual Configure PB" %
%   N25:110  PN5_IE82_BTW_WORD_0  "RIO Rack 0 Slot 2 Analog Input Module BTW to Update Data to Outputs Word 0" %
%   N13:110  PN5_IE82_BTW_DATA  "PN5 RIO Slot 2 Input Configuration Data ma = 0/20madc VDV = 0/10VDV" %
% Rung: 5 %
% his Rung reads the Data from of the 1794-IE8 madc Input Module
% Located in Slot 2 of the Remote I/O Rack Data
% Located in the PN-5 %
SOR XIO N25:110/15 XIO N25:115/15 XIO N25:115/12 OP_D5 0 2 0 N25:115 N12:110 M1:6.300 9 9 3 EOR
%   N25:110/15  PN5_IE82_BTW_ENAB %
%   N25:115/15  PN5_IE82_BTR_ENAB %
%   N25:115/12  PN5_IE82_BTR_ERROR %
%   N25:115  PN5_IE82_BTR_WORD_0  "RIO Rack 0 Slot 2 Analog Input Module BTR to Read Data Word 0" %
%   N12:110  AI109_BIN_DATA %
% Rung: 6 %
% This Rung Reads the Status of the 1794-OE4 madc Output Module
% Located in Slot 3 of the Remote I/O Rack Data
% Located in PN-5 %
SOR XIO N25:125/12 XIO N25:125/13 XIO N25:120/15 OP_D5 0 3 0 N25:125 N12:120 M1:6.400 1 0 3 EOR
%   N25:125/12  PN5_OE41_BTR_ERROR %
%   N25:125/13  PN5_OE41_BTR_DONE %
%   N25:120/15  PN5_OE41_BTW_ENAB %
%   N25:125  PN5_OE41_BTR_WORD_0  "RIO Rack 0 Slot 3 Analog Output Module BTR to Read Status of Outputs Word 0" %
%   N12:120  PN5_OE41_BTR_DATA  "RIO Rack-0, Slot 3 1794-OE4 Status Data" %
% Rung: 7 %
% This Rung Writes Data to the 1794-OE4 madc Output Module
% Located in Slot 3 of the Remote I/O Rack Data
% Located in the PN-5 %
SOR XIO N25:120/12 XIO N25:120/13 OP_D6 0 3 0 N25:120 N13:120 M0:6.400 14 0 3 EOR
%   N25:120/12  PN5_OE41_BTW_ERROR %
%   N25:120/13  PN5_OE41_BTW_DONE %
%   N25:120  PN5_OE41_BTW_WORD_0  "RIO Rack 0 Slot 3 Analog Output Module BTW to Update Data to Outputs Word 0" %
%   N13:120  AO101_BIN_OUTPUT  "AO-101 Rack 0, Slot 3 OE4, Channel 0 Binary Output Data" %

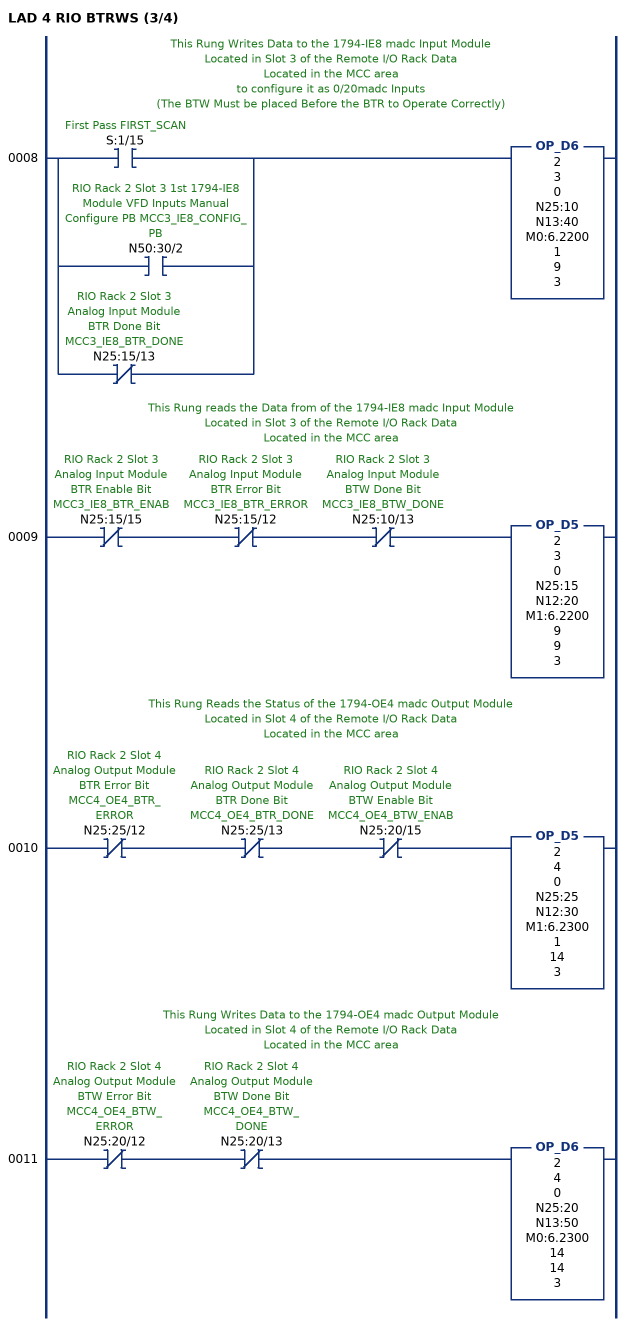
% Rung: 8 %
% This Rung Writes Data to the 1794-IE8 madc Input Module
% Located in Slot 3 of the Remote I/O Rack Data
% Located in the MCC area
% to configure it as 0/20madc Inputs
% 
% (The BTW Must be placed Before the BTR to Operate Correctly) %
SOR BST XIC S:1/15 NXB XIC N50:30/2 NXB XIO N25:15/13 BND OP_D6 2 3 0 N25:10 N13:40 M0:6.2200 1 9 3 EOR
%   S:1/15  FIRST_SCAN  "First Pass" %
%   N50:30/2  MCC3_IE8_CONFIG_PB  "RIO Rack 2 Slot 3 1st 1794-IE8 Module VFD Inputs Manual Configure PB" %
%   N25:15/13  MCC3_IE8_BTR_DONE  "RIO Rack 2 Slot 3 Analog Input Module BTR Done Bit" %
%   N25:10  MCC3_IE8_BTW_WORD_0  "RIO Rack 2 Slot 3 Analog Input Module BTW to Configure Data input" %
%   N13:40  MCC3_IE8_BTW_DATA  "MCC RIO Slot 3 Input Configuration Data ma = 0/20madc VDV = 0/10VDV" %
% Rung: 9 %
% This Rung reads the Data from of the 1794-IE8 madc Input Module
% Located in Slot 3 of the Remote I/O Rack Data
% Located in the MCC area %
SOR XIO N25:15/15 XIO N25:15/12 XIO N25:10/13 OP_D5 2 3 0 N25:15 N12:20 M1:6.2200 9 9 3 EOR
%   N25:15/15  MCC3_IE8_BTR_ENAB  "RIO Rack 2 Slot 3 Analog Input Module BTR Enable Bit" %
%   N25:15/12  MCC3_IE8_BTR_ERROR  "RIO Rack 2 Slot 3 Analog Input Module BTR Error Bit" %
%   N25:10/13  MCC3_IE8_BTW_DONE  "RIO Rack 2 Slot 3 Analog Input Module BTW Done Bit" %
%   N25:15  MCC3_IE8_BTR_WORD_0  "RIO Rack 2 Slot 3 Analog Input Module BTR to Read Status of Inputs" %
%   N12:20  VFD01_BIN_AMPS  "VFD01 Binary Amps" %
% Rung: 10 %
% This Rung Reads the Status of the 1794-OE4 madc Output Module
% Located in Slot 4 of the Remote I/O Rack Data
% Located in the MCC area %
SOR XIO N25:25/12 XIO N25:25/13 XIO N25:20/15 OP_D5 2 4 0 N25:25 N12:30 M1:6.2300 1 14 3 EOR
%   N25:25/12  MCC4_OE4_BTR_ERROR  "RIO Rack 2 Slot 4 Analog Output Module BTR Error Bit" %
%   N25:25/13  MCC4_OE4_BTR_DONE  "RIO Rack 2 Slot 4 Analog Output Module BTR Done Bit" %
%   N25:20/15  MCC4_OE4_BTW_ENAB  "RIO Rack 2 Slot 4 Analog Output Module BTW Enable Bit" %
%   N25:25  MCC4_OE4_BTR_WORD_0  "RIO Rack 2 Slot 4 Analog Output Module BTR to Read Status of Outputs" %
%   N12:30  MCC4_OE4_BTR_DATA  "RIO Rack-2, Slot 4 1794-OE4 Status Data" %
% Rung: 11 %
% This Rung Writes Data to the 1794-OE4 madc Output Module
% Located in Slot 4 of the Remote I/O Rack Data
% Located in the MCC area %
SOR XIO N25:20/12 XIO N25:20/13 OP_D6 2 4 0 N25:20 N13:50 M0:6.2300 14 14 3 EOR
%   N25:20/12  MCC4_OE4_BTW_ERROR  "RIO Rack 2 Slot 4 Analog Output Module BTW Error Bit" %
%   N25:20/13  MCC4_OE4_BTW_DONE  "RIO Rack 2 Slot 4 Analog Output Module BTW Done Bit" %
%   N25:20  MCC4_OE4_BTW_WORD_0  "RIO Rack 2 Slot 4 Analog Output Module BTW to Update Data to Outputs" %
%   N13:50  VFD01_BIN_OUTPUT  "VFD01 Output Binary VFD Speed Signal" %

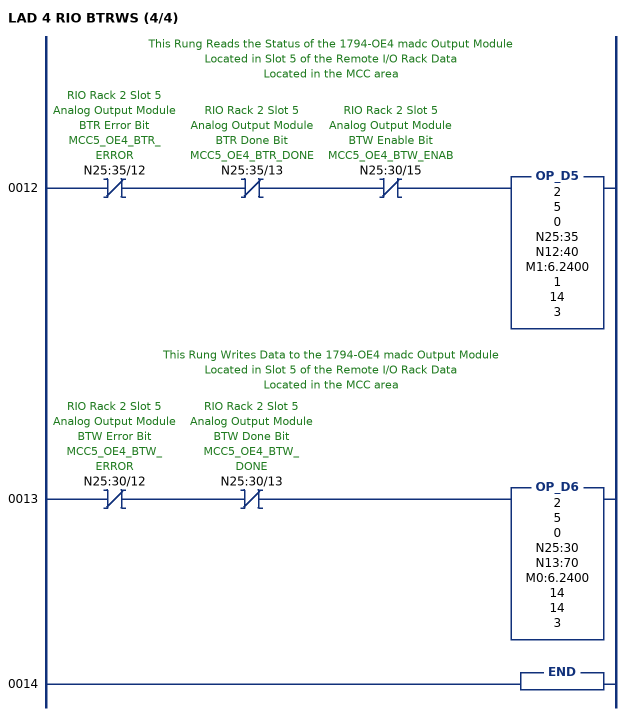
% Rung: 12 %
% This Rung Reads the Status of the 1794-OE4 madc Output Module
% Located in Slot 5 of the Remote I/O Rack Data
% Located in the MCC area %
SOR XIO N25:35/12 XIO N25:35/13 XIO N25:30/15 OP_D5 2 5 0 N25:35 N12:40 M1:6.2400 1 14 3 EOR
%   N25:35/12  MCC5_OE4_BTR_ERROR  "RIO Rack 2 Slot 5 Analog Output Module BTR Error Bit" %
%   N25:35/13  MCC5_OE4_BTR_DONE  "RIO Rack 2 Slot 5 Analog Output Module BTR Done Bit" %
%   N25:30/15  MCC5_OE4_BTW_ENAB  "RIO Rack 2 Slot 5 Analog Output Module BTW Enable Bit" %
%   N25:35  MCC5_OE4_BTR_WORD_0  "RIO Rack 2 Slot 5 Analog Output Module BTR to Read Status of Outputs" %
%   N12:40  MCC5_OE4_BTR_DATA  "RIO Rack-2, Slot 5 1794-OE4 Status Data" %
% Rung: 13 %
% This Rung Writes Data to the 1794-OE4 madc Output Module
% Located in Slot 5 of the Remote I/O Rack Data
% Located in the MCC area %
SOR XIO N25:30/12 XIO N25:30/13 OP_D6 2 5 0 N25:30 N13:70 M0:6.2400 14 14 3 EOR
%   N25:30/12  MCC5_OE4_BTW_ERROR  "RIO Rack 2 Slot 5 Analog Output Module BTW Error Bit" %
%   N25:30/13  MCC5_OE4_BTW_DONE  "RIO Rack 2 Slot 5 Analog Output Module BTW Done Bit" %
%   N25:30  MCC5_OE4_BTW_WORD_0  "RIO Rack 2 Slot 5 Analog Output Module BTW to Update Data to Outputs" %
%   N13:70  VFD05_BIN_OUTPUT  "VFD05 Output Binary VFD Speed Signal" %
% Rung: 14 %
SOR END EOR

LADDER 10 "ALARM CTRL"    % Alarm Controls %
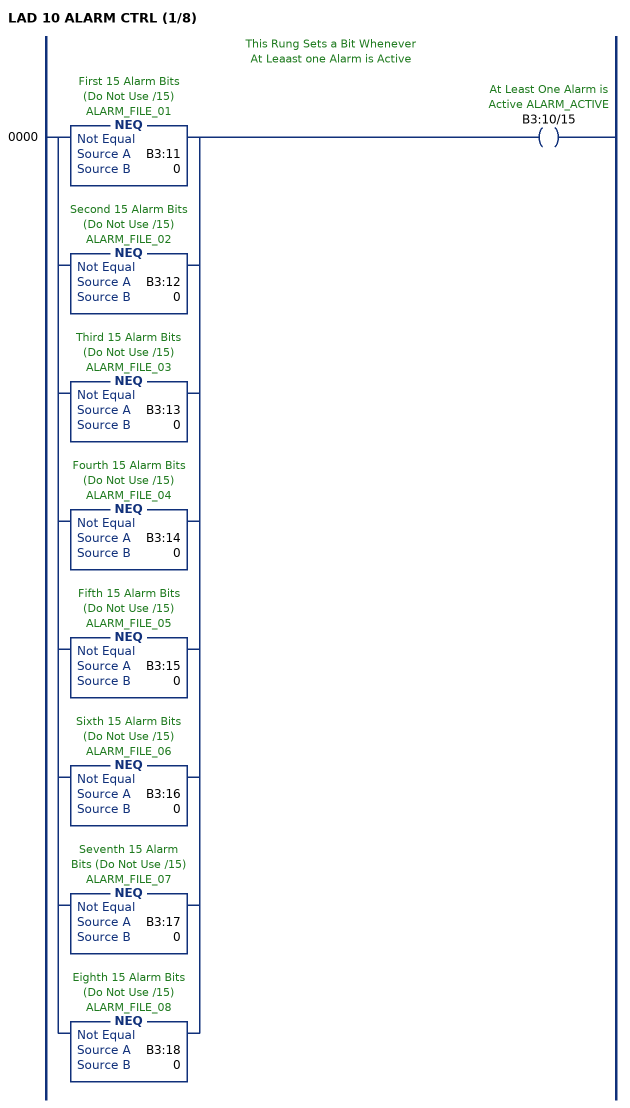
% Rung: 0 %
% This Rung Sets a Bit Whenever
% At Leaast one Alarm is Active %
SOR BST NEQ B3:11 0 NXB NEQ B3:12 0 NXB NEQ B3:13 0 NXB NEQ B3:14 0 NXB NEQ B3:15 0 NXB NEQ B3:16 0 NXB NEQ B3:17 0 NXB NEQ B3:18 0 BND OTE B3:10/15 EOR
%   B3:11  ALARM_FILE_01  "First 15 Alarm Bits (Do Not Use /15)" %
%   B3:12  ALARM_FILE_02  "Second 15 Alarm Bits (Do Not Use /15)" %
%   B3:13  ALARM_FILE_03  "Third 15 Alarm Bits (Do Not Use /15)" %
%   B3:14  ALARM_FILE_04  "Fourth 15 Alarm Bits (Do Not Use /15)" %
%   B3:15  ALARM_FILE_05  "Fifth 15 Alarm Bits (Do Not Use /15)" %
%   B3:16  ALARM_FILE_06  "Sixth 15 Alarm Bits (Do Not Use /15)" %
%   B3:17  ALARM_FILE_07  "Seventh 15 Alarm Bits (Do Not Use /15)" %
%   B3:18  ALARM_FILE_08  "Eighth 15 Alarm Bits (Do Not Use /15)" %
%   B3:10/15  ALARM_ACTIVE  "At Least One Alarm is Active" %

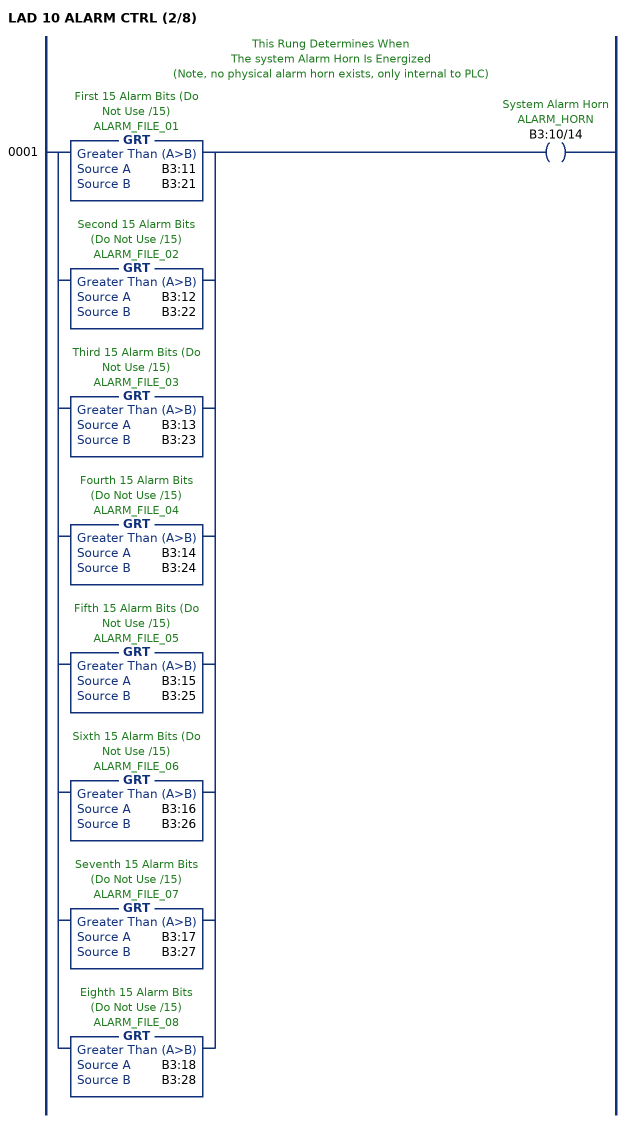
% Rung: 1 %
% This Rung Determines When
% The system Alarm Horn Is Energized
% (Note, no physical alarm horn exists, only internal to PLC) %
SOR BST GRT B3:11 B3:21 NXB GRT B3:12 B3:22 NXB GRT B3:13 B3:23 NXB GRT B3:14 B3:24 NXB GRT B3:15 B3:25 NXB GRT B3:16 B3:26 NXB GRT B3:17 B3:27 NXB GRT B3:18 B3:28 BND OTE B3:10/14 EOR
%   B3:11  ALARM_FILE_01  "First 15 Alarm Bits (Do Not Use /15)" %
%   B3:21  ALARM_FILE_01_ACK  "First 15 Alarm Acknowledge Bits" %
%   B3:12  ALARM_FILE_02  "Second 15 Alarm Bits (Do Not Use /15)" %
%   B3:22  ALARM_FILE_02_ACK  "First 15 Alarm Acknowledge Bits" %
%   B3:13  ALARM_FILE_03  "Third 15 Alarm Bits (Do Not Use /15)" %
%   B3:23  ALARM_FILE_03_ACK  "First 15 Alarm Acknowledge Bits" %
%   B3:14  ALARM_FILE_04  "Fourth 15 Alarm Bits (Do Not Use /15)" %
%   B3:24  ALARM_FILE_04_ACK  "First 15 Alarm Acknowledge Bits" %
%   B3:15  ALARM_FILE_05  "Fifth 15 Alarm Bits (Do Not Use /15)" %
%   B3:25  ALARM_FILE_05_ACK  "First 15 Alarm Acknowledge Bits" %
%   B3:16  ALARM_FILE_06  "Sixth 15 Alarm Bits (Do Not Use /15)" %
%   B3:26  ALARM_FILE_06_ACK  "Sixth 15 Alarm Acknowledge Bits" %
%   B3:17  ALARM_FILE_07  "Seventh 15 Alarm Bits (Do Not Use /15)" %
%   B3:27  ALARM_FILE_07_ACK  "Seventh 15 Alarm Acknowledge Bits" %
%   B3:18  ALARM_FILE_08  "Eighth 15 Alarm Bits (Do Not Use /15)" %
%   B3:28  ALARM_FILE_08_ACK  "Eighth 15 Alarm Acknowledge Bits" %
%   B3:10/14  ALARM_HORN  "System Alarm Horn" %

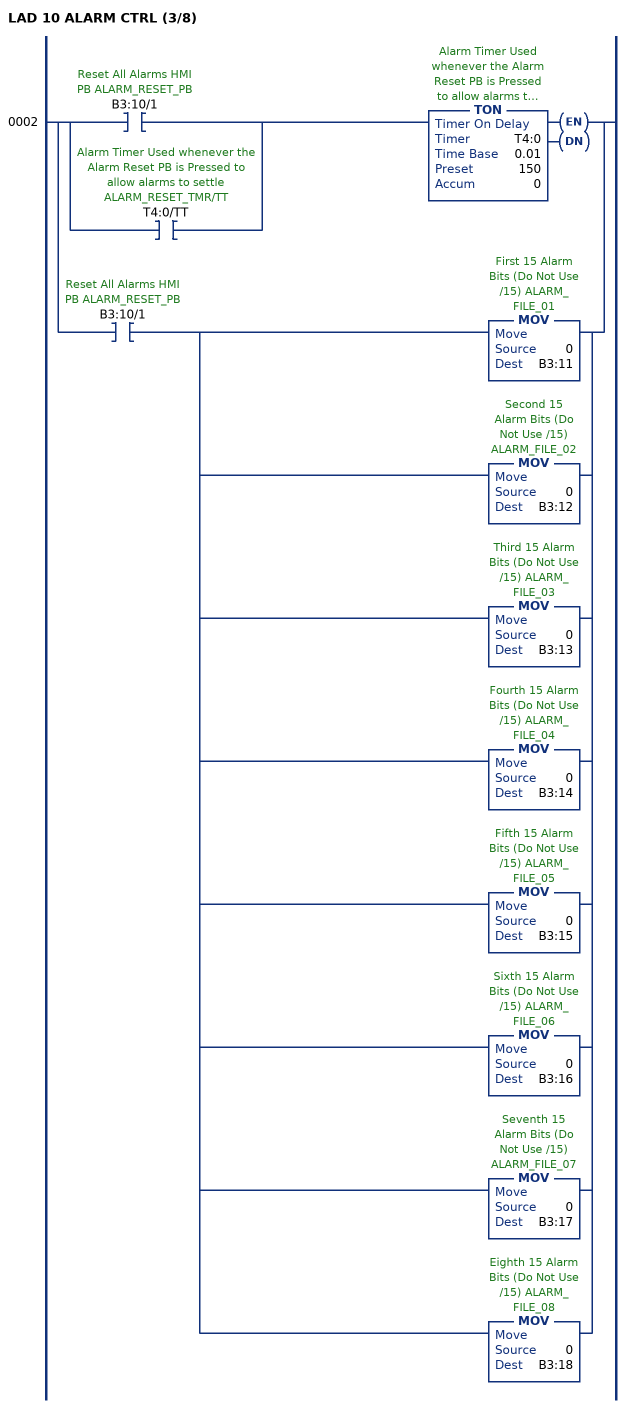
% Rung: 2 %
SOR BST BST XIC B3:10/1 NXB XIC T4:0/TT BND TON T4:0 0.01 150 0 NXB XIC B3:10/1 BST MOV 0 B3:11 NXB MOV 0 B3:12 NXB MOV 0 B3:13 NXB MOV 0 B3:14 NXB MOV 0 B3:15 NXB MOV 0 B3:16 NXB MOV 0 B3:17 NXB MOV 0 B3:18 BND BND EOR
%   B3:10/1  ALARM_RESET_PB  "Reset All Alarms HMI PB" %
%   T4:0  ALARM_RESET_TMR  "Alarm Timer Used whenever the Alarm Reset PB is Pressed to allow alarms to settle" %
%   B3:11  ALARM_FILE_01  "First 15 Alarm Bits (Do Not Use /15)" %
%   B3:12  ALARM_FILE_02  "Second 15 Alarm Bits (Do Not Use /15)" %
%   B3:13  ALARM_FILE_03  "Third 15 Alarm Bits (Do Not Use /15)" %
%   B3:14  ALARM_FILE_04  "Fourth 15 Alarm Bits (Do Not Use /15)" %
%   B3:15  ALARM_FILE_05  "Fifth 15 Alarm Bits (Do Not Use /15)" %
%   B3:16  ALARM_FILE_06  "Sixth 15 Alarm Bits (Do Not Use /15)" %
%   B3:17  ALARM_FILE_07  "Seventh 15 Alarm Bits (Do Not Use /15)" %
%   B3:18  ALARM_FILE_08  "Eighth 15 Alarm Bits (Do Not Use /15)" %

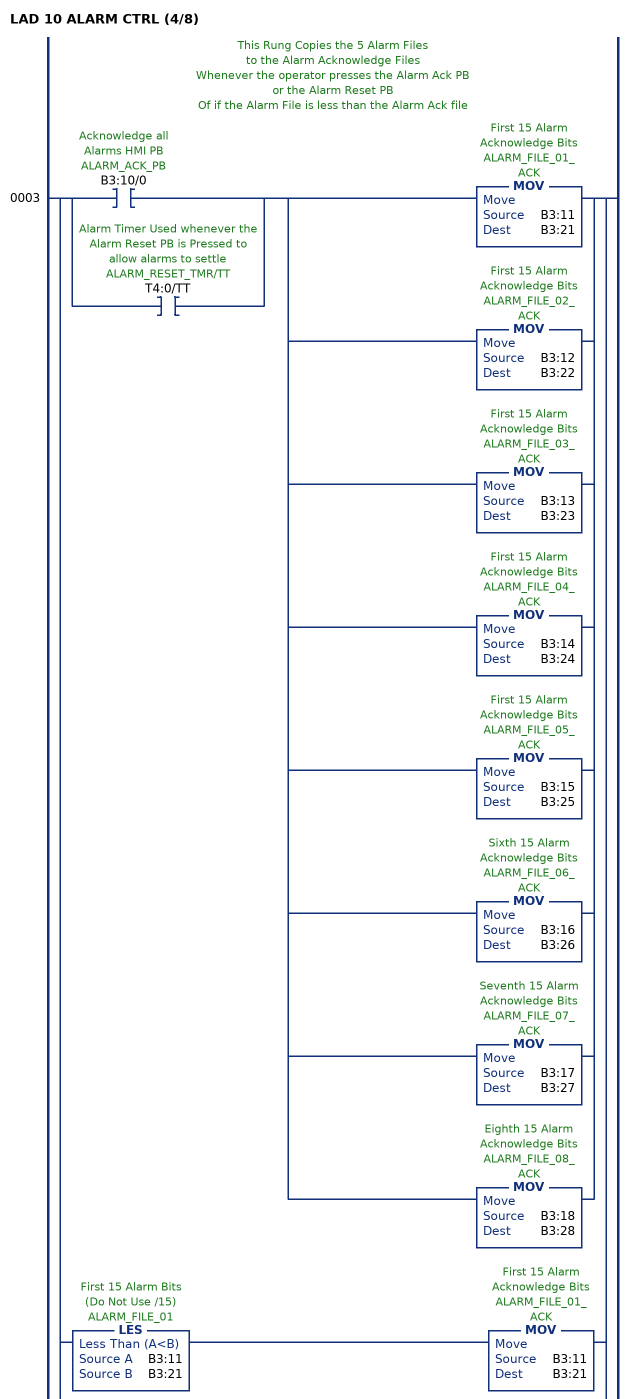

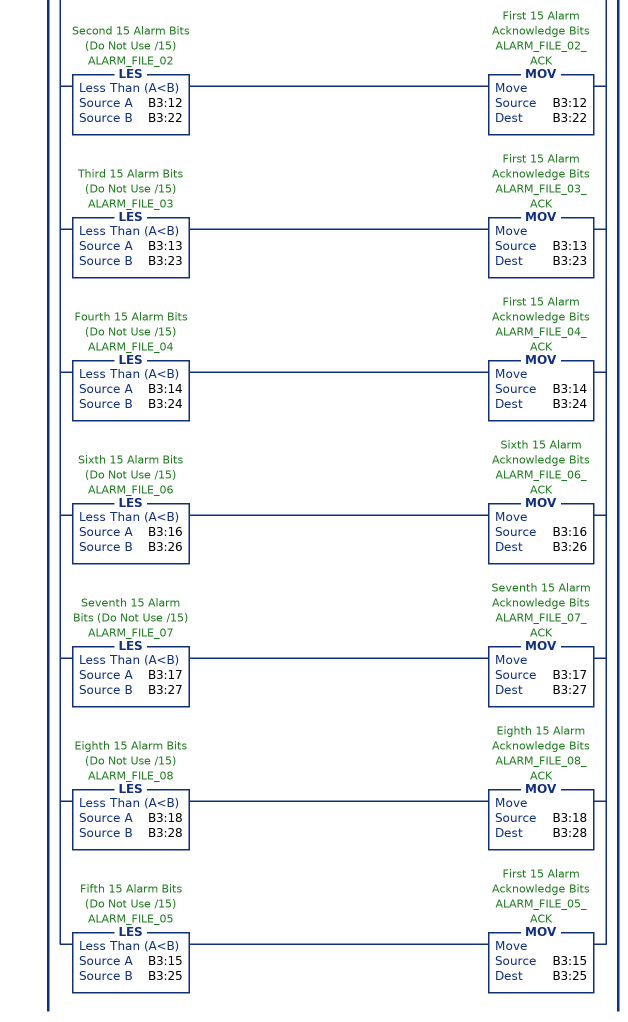
% Rung: 3 %
% This Rung Copies the 5 Alarm Files
% to the Alarm Acknowledge Files
% Whenever the operator presses the Alarm Ack PB
% or the Alarm Reset PB
% Of if the Alarm File is less than the Alarm Ack file %
SOR BST BST XIC B3:10/0 NXB XIC T4:0/TT BND BST MOV B3:11 B3:21 NXB MOV B3:12 B3:22 NXB MOV B3:13 B3:23 NXB MOV B3:14 B3:24 NXB MOV B3:15 B3:25 NXB MOV B3:16 B3:26 NXB MOV B3:17 B3:27 NXB MOV B3:18 B3:28 BND NXB LES B3:11 B3:21 MOV B3:11 B3:21 NXB LES B3:12 B3:22 MOV B3:12 B3:22 NXB LES B3:13 B3:23 MOV B3:13 B3:23 NXB LES B3:14 B3:24 MOV B3:14 B3:24 NXB LES B3:16 B3:26 MOV B3:16 B3:26 NXB LES B3:17 B3:27 MOV B3:17 B3:27 NXB LES B3:18 B3:28 MOV B3:18 B3:28 NXB LES B3:15 B3:25 MOV B3:15 B3:25 BND EOR
%   B3:10/0  ALARM_ACK_PB  "Acknowledge all Alarms HMI PB" %
%   T4:0  ALARM_RESET_TMR  "Alarm Timer Used whenever the Alarm Reset PB is Pressed to allow alarms to settle" %
%   B3:11  ALARM_FILE_01  "First 15 Alarm Bits (Do Not Use /15)" %
%   B3:21  ALARM_FILE_01_ACK  "First 15 Alarm Acknowledge Bits" %
%   B3:12  ALARM_FILE_02  "Second 15 Alarm Bits (Do Not Use /15)" %
%   B3:22  ALARM_FILE_02_ACK  "First 15 Alarm Acknowledge Bits" %
%   B3:13  ALARM_FILE_03  "Third 15 Alarm Bits (Do Not Use /15)" %
%   B3:23  ALARM_FILE_03_ACK  "First 15 Alarm Acknowledge Bits" %
%   B3:14  ALARM_FILE_04  "Fourth 15 Alarm Bits (Do Not Use /15)" %
%   B3:24  ALARM_FILE_04_ACK  "First 15 Alarm Acknowledge Bits" %
%   B3:15  ALARM_FILE_05  "Fifth 15 Alarm Bits (Do Not Use /15)" %
%   B3:25  ALARM_FILE_05_ACK  "First 15 Alarm Acknowledge Bits" %
%   B3:16  ALARM_FILE_06  "Sixth 15 Alarm Bits (Do Not Use /15)" %
%   B3:26  ALARM_FILE_06_ACK  "Sixth 15 Alarm Acknowledge Bits" %
%   B3:17  ALARM_FILE_07  "Seventh 15 Alarm Bits (Do Not Use /15)" %
%   B3:27  ALARM_FILE_07_ACK  "Seventh 15 Alarm Acknowledge Bits" %
%   B3:18  ALARM_FILE_08  "Eighth 15 Alarm Bits (Do Not Use /15)" %
%   B3:28  ALARM_FILE_08_ACK  "Eighth 15 Alarm Acknowledge Bits" %

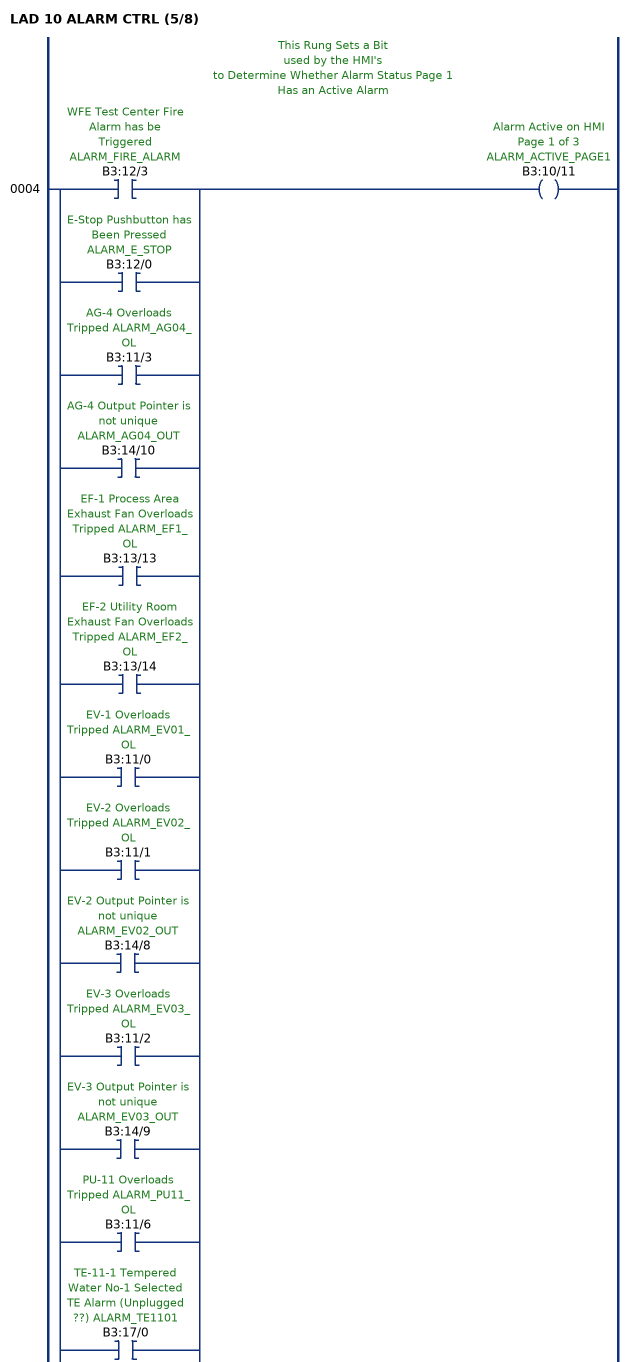

